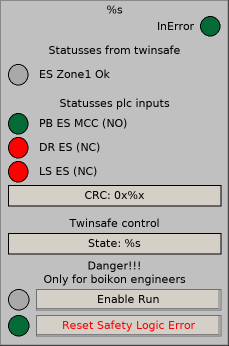
VISUALIZATION Vis_SafetyZone1  // 229x346
VAR_INPUT
	I_Title:string;
END_VAR

VAR_IN_OUT
	IO_SafetyLogic:cntrl_SafetyGroup1;
END_VAR
    Rectangle (0,0 229x346)
    Rectangle (12,0 205x20), "%s", text variable: I_Title
    Rectangle (8,233 213x21), "State: %s", text variable: IO_SafetyLogic.eS
    Button (36,315 185x21), "Reset Safety Logic Error", pressed state: IO_SafetyLogic.PbSf_ResetSafetyErrors.P_BypassStateTrue
        tap IO_SafetyLogic.PbSf_ResetSafetyErrors.P_BypassStateTrue
    Ellipse (8,315 21x21), colour toggle: IO_SafetyLogic.HMI.STS.LogicInError
    Ellipse (8,289 21x21), colour toggle: IO_SafetyLogic.Isf_STS_SafetyInRun.HMI.STS.State
    Rectangle (8,257 213x31), "Danger!!! Only for boikon engineers"
    Button (36,289 185x21), "Enable Run", pressed state: IO_SafetyLogic.HMI.STS.PB_RunSafetyLogic
        toggle IO_SafetyLogic.HMI.STS.PB_RunSafetyLogic
    Ellipse (8,64 20x21), colour toggle: IO_SafetyLogic.Isf_STS_ES_Zone1_OK.HMI.STS.State
    Rectangle (36,64 181x21), "ES Zone1 Ok"
    Ellipse (8,113 20x21), colour toggle: IO_SafetyLogic.PB_ES_MainCabinet.HMI.STS.State
    Rectangle (36,113 181x21), "PB ES MCC (NO)"
    Ellipse (8,137 20x21), colour toggle: IO_SafetyLogic.DR_Front.HMI.STS.State
    Rectangle (36,137 181x21), "DR ES (NC)"
    Ellipse (8,161 20x21), colour toggle: IO_SafetyLogic.LS_Entry1.HMI.STS.State
    Rectangle (36,161 181x21), "LS ES (NC)"
    Ellipse (200,16 20x20), colour toggle: IO_SafetyLogic.HMI.P_STS_InError
    Rectangle (128,16 69x21), "InError"
    Label (8,40 213x21), "Statusses from twinsafe"
    Label (8,93 213x21), "Statusses plc inputs"
    Label (8,213 213x21), "Twinsafe control"
    Rectangle (8,185 213x21), "CRC: 0x%x", text variable: IO_SafetyLogic.HMI.STS.CrcCodeProject
END_VISUALIZATION

(* stored: Version 1.1.0.1
   Visu Vis_SafetyZone1: Id {5a4749fc-7e5d-02c1-105b-1be2175978d8} *)
